INTERFACE ITF_DeviceStatus

PROPERTY Faults : STRING
GET
END_GET
END_PROPERTY

PROPERTY StatusOK : BOOL
GET
END_GET
END_PROPERTY

END_INTERFACE

(* stored: Version 1.1.0.1, ProductVersion 3.1.4024.12
   Itf ITF_DeviceStatus: Id {6da6c48b-bf2a-4da2-b6f4-ca51580f04b7}
   Property Faults: Id {9e21ca3e-a1a5-45d4-9aa9-43b8ad738a3a}
   Get Get: Id {3d92b4a5-df9d-45d2-9167-e91d5a9523fa}
   Property StatusOK: Id {c6774711-ac1e-4ada-bd1a-7ddfa18eab87}
   Get Get: Id {3f9e73b5-1a0c-4c18-8573-f3f1fb0992f3} *)
